// Mitsubishi GX Works2 project: 2023-04-20 #2   PLC: Q03UDV

// global labels: Global1
VAR_GLOBAL
  PB1 AT X0 : BOOL;
  PB2 AT X1 : BOOL;
  정지 AT X2 : BOOL;
  공급후진 AT X3 : BOOL;
  공급전진 AT X4 : BOOL;
  가공후진 AT X5 : BOOL;
  가공전진 AT X6 : BOOL;
  송출후진 AT X7 : BOOL;
  송출전진 AT X8 : BOOL;
  배출후진 AT X9 : BOOL;
  배출전진 AT X0A : BOOL;
  매거진 AT X0B : BOOL;
  가공센서 AT X0C : BOOL;
  송출센서 AT X0D : BOOL;
  비금속센서 AT X0E : BOOL;
  금속센서 AT X0F : BOOL;
  PB3 AT X10 : BOOL;
  적색 AT Y20 : BOOL;
  황색 AT Y21 : BOOL;
  녹색 AT Y22 : BOOL;
  공급1 AT Y23 : BOOL;
  공급2 AT Y24 : BOOL;
  가공 AT Y25 : BOOL;
  드릴 AT Y26 : BOOL;
  송출 AT Y27 : BOOL;
  배출 AT Y28 : BOOL;
  컨베이어 AT Y29 : BOOL;
END_VAR

PROGRAM 기본동작
VAR
  STATE : INT;
END_VAR
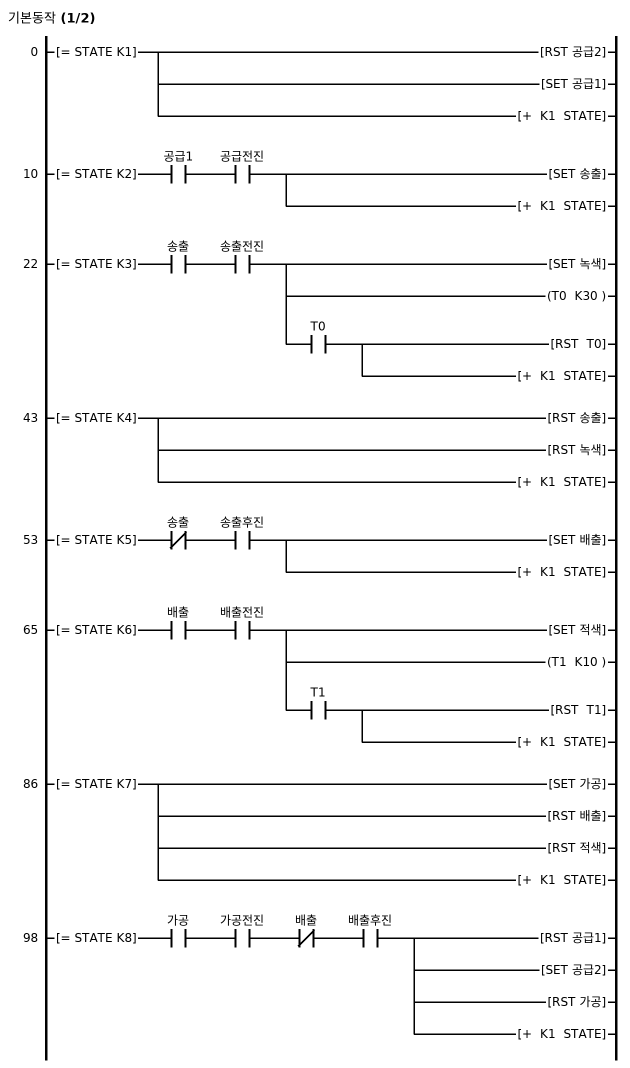
0     LD=     STATE K1
      RST     공급2
      SET     공급1
      +       K1 STATE
10    LD=     STATE K2
      AND     공급1
      AND     공급전진
      SET     송출
      +       K1 STATE
22    LD=     STATE K3
      AND     송출
      AND     송출전진
      SET     녹색
      OUT     T0 K30
      AND     T0
      RST     T0
      +       K1 STATE
43    LD=     STATE K4
      RST     송출
      RST     녹색
      +       K1 STATE
53    LD=     STATE K5
      ANI     송출
      AND     송출후진
      SET     배출
      +       K1 STATE
65    LD=     STATE K6
      AND     배출
      AND     배출전진
      SET     적색
      OUT     T1 K10
      AND     T1
      RST     T1
      +       K1 STATE
86    LD=     STATE K7
      SET     가공
      RST     배출
      RST     적색
      +       K1 STATE
98    LD=     STATE K8
      AND     가공
      AND     가공전진
      ANI     배출
      AND     배출후진
      RST     공급1
      SET     공급2
      RST     가공
      +       K1 STATE
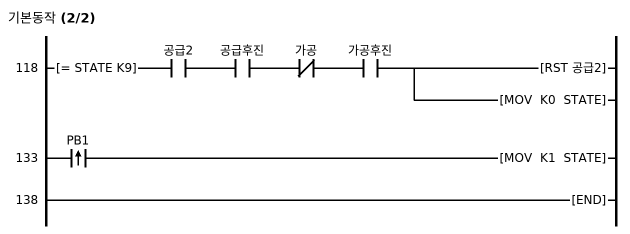
118   LD=     STATE K9
      AND     공급2
      AND     공급후진
      ANI     가공
      AND     가공후진
      RST     공급2
      MOV     K0 STATE
133   LDP     PB1
      MOV     K1 STATE
138   END
END_PROGRAM

PROGRAM 응용동작1
VAR
  STATE : INT;
END_VAR
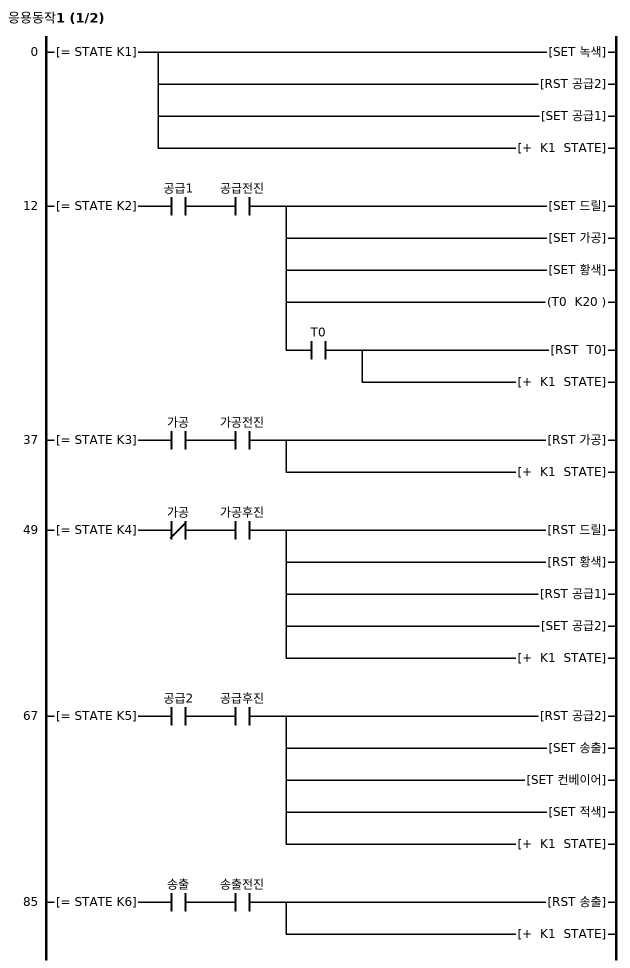
0     LD=     STATE K1
      SET     녹색
      RST     공급2
      SET     공급1
      +       K1 STATE
12    LD=     STATE K2
      AND     공급1
      AND     공급전진
      SET     드릴
      SET     가공
      SET     황색
      OUT     T0 K20
      AND     T0
      RST     T0
      +       K1 STATE
37    LD=     STATE K3
      AND     가공
      AND     가공전진
      RST     가공
      +       K1 STATE
49    LD=     STATE K4
      ANI     가공
      AND     가공후진
      RST     드릴
      RST     황색
      RST     공급1
      SET     공급2
      +       K1 STATE
67    LD=     STATE K5
      AND     공급2
      AND     공급후진
      RST     공급2
      SET     송출
      SET     컨베이어
      SET     적색
      +       K1 STATE
85    LD=     STATE K6
      AND     송출
      AND     송출전진
      RST     송출
      +       K1 STATE
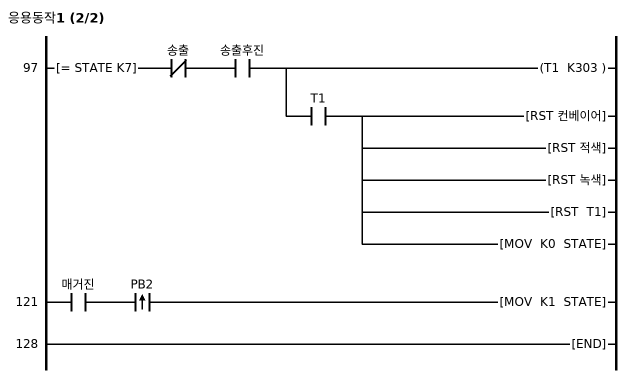
97    LD=     STATE K7
      ANI     송출
      AND     송출후진
      OUT     T1 K303
      AND     T1
      RST     컨베이어
      RST     적색
      RST     녹색
      RST     T1
      MOV     K0 STATE
121   LD      매거진
      ANDP    PB2
      MOV     K1 STATE
128   END
END_PROGRAM

PROGRAM 응용동작2
VAR
  STATE : INT;
  MAGAZINE : INT;
END_VAR
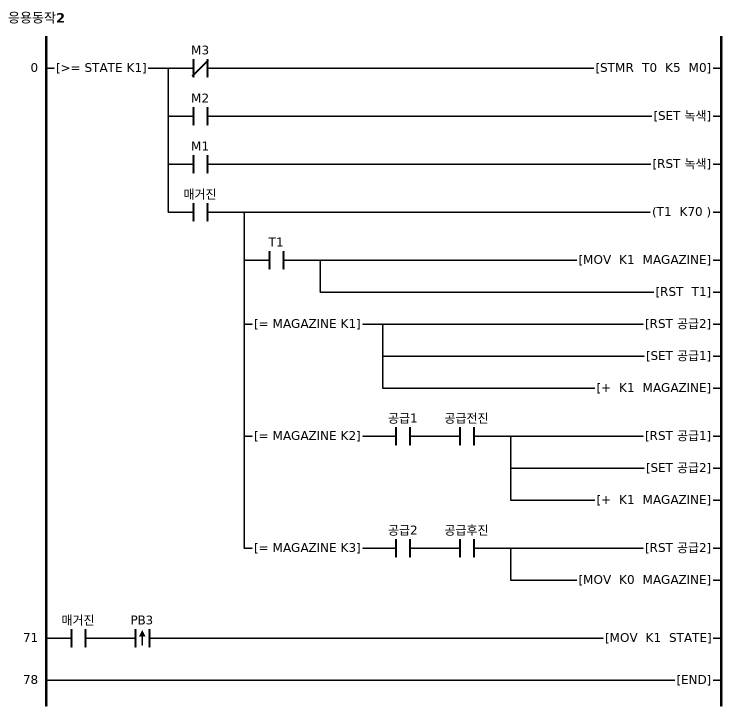
0     LD>=    STATE K1
      MPS
      ANI     M3
      STMR    T0 K5 M0
      MRD
      AND     M2
      SET     녹색
      MRD
      AND     M1
      RST     녹색
      MPP
      AND     매거진
      OUT     T1 K70
      MPS
      AND     T1
      MOV     K1 MAGAZINE
      RST     T1
      MRD
      AND=    MAGAZINE K1
      RST     공급2
      SET     공급1
      +       K1 MAGAZINE
      MRD
      AND=    MAGAZINE K2
      AND     공급1
      AND     공급전진
      RST     공급1
      SET     공급2
      +       K1 MAGAZINE
      MPP
      AND=    MAGAZINE K3
      AND     공급2
      AND     공급후진
      RST     공급2
      MOV     K0 MAGAZINE
71    LD      매거진
      ANDP    PB3
      MOV     K1 STATE
78    END
END_PROGRAM
